ABB RAPID module: SERVER.mod

MODULE SERVER

!////////////////
!GLOBAL VARIABLES
!////////////////

!//Robot configuration
PERS tooldata currentTool := [TRUE,[[0,0,0],[-0.27065,0.65328,-0.2706,0.65328]],[0.001,[0,0,0.001],[1,0,0,0],0,0,0]];
PERS wobjdata currentWobj := [FALSE,TRUE,"",[[0,0,0],[1,0,0,0]],[[0,0,0],[1,0,0,0]]];
PERS speeddata currentSpeed;
PERS zonedata currentZone;

!// Clock Synchronization
PERS bool startLog:=TRUE;
PERS bool startRob:=TRUE;

!// Mutex between logger and changing the tool and work objects
PERS bool frameMutex:=FALSE;

!//PC communication
VAR socketdev clientSocket;
VAR socketdev serverSocket;
VAR num instructionCode;
VAR num params{10};
VAR num nParams;

PERS string ipController:= "20.20.20.21"; !robot default IP
!PERS string ipController:= "127.0.0.1"; !local IP for testing in simulation
PERS num serverPort:= 5000;

!//Motion of the robot
VAR robtarget cartesianTarget;
VAR jointtarget jointsTarget;
VAR bool moveCompleted; !Set to true after finishing a Move instruction.

!//Buffered move variables
CONST num MAX_BUFFER := 128;
PERS bool paused := FALSE;
PERS num BUFFER_POS;
PERS num BUFFER_LEFT;
PERS bool MOVING;
PERS robtarget bufferTargets{MAX_BUFFER};
PERS speeddata bufferSpeeds{MAX_BUFFER};
PERS bool BUFFER_LOCKED;

!//External axis position variables
PERS extjoint externalAxis;

!//Circular move buffer
VAR robtarget circPoint;

!//Correct Instruction Execution and possible return values
VAR num ok;
CONST num SERVER_BAD_MSG :=  0;
CONST num SERVER_OK := 1;




!////////////////
!LOCAL METHODS
!////////////////

!//Method to parse the message received from a PC
!// If correct message, loads values on:
!// - instructionCode.
!// - nParams: Number of received parameters.
!// - params{nParams}: Vector of received params.
PROC ParseMsg(string msg)
    !//Local variables
    VAR bool auxOk;
    VAR num ind:=1;
    VAR num newInd;
    VAR num length;
    VAR num indParam:=1;
    VAR string subString;
    VAR bool end := FALSE;

    !//Find the end character
    length := StrMatch(msg,1,"#");
    IF length > StrLen(msg) THEN
        !//Corrupt message
        nParams := -1;
    ELSE
        !//Read Instruction code
        newInd := StrMatch(msg,ind," ") + 1;
        subString := StrPart(msg,ind,newInd - ind - 1);
        auxOk:= StrToVal(subString, instructionCode);
        IF auxOk = FALSE THEN
            !//Impossible to read instruction code
            nParams := -1;
        ELSE
            ind := newInd;
            !//Read all instruction parameters (maximum of 8)
            WHILE end = FALSE DO
                newInd := StrMatch(msg,ind," ") + 1;
                IF newInd > length THEN
                    end := TRUE;
                ELSE
                    subString := StrPart(msg,ind,newInd - ind - 1);
                    auxOk := StrToVal(subString, params{indParam});
                    indParam := indParam + 1;
                    ind := newInd;
                ENDIF
            ENDWHILE
            nParams:= indParam - 1;
        ENDIF
    ENDIF
ENDPROC


!//Handshake between server and client:
!// - Creates socket.
!// - Waits for incoming TCP connection.
PROC ServerCreateAndConnect(string ip, num port)
    VAR string clientIP;

    SocketCreate serverSocket;
    SocketBind serverSocket, ip, port;
    SocketListen serverSocket;
    TPWrite "SERVER: Server waiting for incoming connections ...";
    WHILE SocketGetStatus(clientSocket) <> SOCKET_CONNECTED DO
        SocketAccept serverSocket,clientSocket \ClientAddress:=clientIP \Time:=WAIT_MAX;
        IF SocketGetStatus(clientSocket) <> SOCKET_CONNECTED THEN
            TPWrite "SERVER: Problem serving an incoming connection.";
            TPWrite "SERVER: Try reconnecting.";
        ENDIF
        !//Wait 0.5 seconds for the next reconnection
        WaitTime 0.5;
    ENDWHILE
    TPWrite "SERVER: Connected to IP " + clientIP;
ENDPROC


!//Parameter initialization
!// Loads default values for
!// - Tool.
!// - WorkObject.
!// - Zone.
!// - Speed.
PROC Initialize()
    currentTool := [TRUE,[[0,0,0],[1,0,0,0]],[0.001,[0,0,0.001],[1,0,0,0],0,0,0]];
    currentWobj := [FALSE,TRUE,"",[[0,0,0],[1,0,0,0]],[[0,0,0],[1,0,0,0]]];
    currentSpeed := [250, 250, 250, 250];
    currentZone := [FALSE, 0.3, 0.3,0.3,0.03,0.3,0.03]; !z0

	!Find the current external axis values so they don't move when we start
	jointsTarget := CJointT();
	externalAxis := jointsTarget.extax;
ENDPROC


!////////////////////////
!//SERVER: Main procedure
!////////////////////////
PROC main()
    !//Local variables
    VAR string receivedString;   !//Received string
    VAR string sendString;       !//Reply string
    VAR string addString;        !//String to add to the reply.
    VAR bool connected;          !//Client connected
    VAR bool reconnected;        !//Drop and reconnection happened during serving a command
    VAR robtarget cartesianPose;
    VAR jointtarget jointsPose;

    VAR robtarget pwobj1;
    VAR robtarget pwobj2;
    VAR robtarget pwobj3;
    VAR wobjdata cwobj;
    VAR num writePos := 1;

    VAR num speed := 250;
    VAR speeddata newSpeed;


    !//Motion configuration
    !ConfL \Off;
    !SingArea \Wrist;
    moveCompleted:= TRUE;

    !//Initialization of WorkObject, Tool, Speed and Zone
    Initialize;

    !//Socket connection
    connected:=FALSE;
    ServerCreateAndConnect ipController,serverPort;
    connected:=TRUE;

    !//Server Loop
    WHILE TRUE DO
        !//Initialization of program flow variables
        ok:=SERVER_OK;              !//Correctness of executed instruction.
        reconnected:=FALSE;         !//Has communication dropped after receiving a command?
        addString := "";

        !//Wait for a command
        SocketReceive clientSocket \Str:=receivedString  \ReadNoOfBytes:=76 \Time:=WAIT_MAX;
        ParseMsg receivedString;

        !//Execution of the command
        TEST instructionCode
            CASE 0: !Ping
                IF nParams = 0 THEN
                    ok := SERVER_OK;
                ELSE
                    ok := SERVER_BAD_MSG;
                ENDIF

!            CASE 1: !Cartesian Move
!                IF nParams = 7 THEN
!                    cartesianTarget :=[[params{1},params{2},params{3}],
!                                       [params{4},params{5},params{6},params{7}],
!                                       [0,0,0,0],
!                                       externalAxis];
!                    ok := SERVER_OK;
!                    moveCompleted := FALSE;
!                    MoveL cartesianTarget, currentSpeed, currentZone, currentTool \WObj:=currentWobj ;
!                    moveCompleted := TRUE;
!                ELSE
!                    ok := SERVER_BAD_MSG;
!                ENDIF

!            CASE 2: !Joint Move
!                IF nParams = 6 THEN
!                    jointsTarget:=[[params{1},params{2},params{3},params{4},params{5},params{6}], externalAxis];
!                    ok := SERVER_OK;
!                    moveCompleted := FALSE;
!                    MoveAbsJ jointsTarget, currentSpeed, currentZone, currentTool \Wobj:=currentWobj;
!                    moveCompleted := TRUE;
!                ELSE
!                    ok :=SERVER_BAD_MSG;
!                ENDIF

            CASE 3: !Get Cartesian Coordinates (with current tool and workobject)
                IF nParams = 0 THEN
                    cartesianPose := CRobT(\Tool:=currentTool \WObj:=currentWObj);
                    addString := NumToStr(cartesianPose.trans.x,2) + " ";
                    addString := addString + NumToStr(cartesianPose.trans.y,2) + " ";
                    addString := addString + NumToStr(cartesianPose.trans.z,2) + " ";
                    addString := addString + NumToStr(cartesianPose.rot.q1,3) + " ";
                    addString := addString + NumToStr(cartesianPose.rot.q2,3) + " ";
                    addString := addString + NumToStr(cartesianPose.rot.q3,3) + " ";
                    addString := addString + NumToStr(cartesianPose.rot.q4,3); !End of string
                    ok := SERVER_OK;
                ELSE
                    ok :=SERVER_BAD_MSG;
                ENDIF

            CASE 4: !Get Joint Coordinates
                IF nParams = 0 THEN
                    jointsPose := CJointT();
                    addString := NumToStr(jointsPose.robax.rax_1,2) + " ";
                    addString := addString + NumToStr(jointsPose.robax.rax_2,2) + " ";
                    addString := addString + NumToStr(jointsPose.robax.rax_3,2) + " ";
                    addString := addString + NumToStr(jointsPose.robax.rax_4,2) + " ";
                    addString := addString + NumToStr(jointsPose.robax.rax_5,2) + " ";
                    addString := addString + NumToStr(jointsPose.robax.rax_6,2); !End of string
                    ok := SERVER_OK;
                ELSE
                    ok:=SERVER_BAD_MSG;
                ENDIF
			CASE 5: !Get external axis positions
                IF nParams = 0 THEN
                    jointsPose := CJointT();
                    addString := StrPart(NumToStr(jointsTarget.extax.eax_a, 2),1,8) + " ";
                    addString := addString + StrPart(NumToStr(jointsTarget.extax.eax_b,2),1,8) + " ";
                    addString := addString + StrPart(NumToStr(jointsTarget.extax.eax_c,2),1,8) + " ";
                    addString := addString + StrPart(NumToStr(jointsTarget.extax.eax_d,2),1,8) + " ";
                    addString := addString + StrPart(NumToStr(jointsTarget.extax.eax_e,2),1,8) + " ";
                    addString := addString + StrPart(NumToStr(jointsTarget.extax.eax_f,2),1,8); !End of string
                    ok := SERVER_OK;
                ELSE
                    ok:=SERVER_BAD_MSG;
                ENDIF

            CASE 6: !Set Tool
                IF nParams = 7 THEN
		   WHILE (frameMutex) DO
		        WaitTime .01; !// If the frame is being used by logger, wait here
		   ENDWHILE
		frameMutex:= TRUE;
                    currentTool.tframe.trans.x:=params{1};
                    currentTool.tframe.trans.y:=params{2};
                    currentTool.tframe.trans.z:=params{3};
                    currentTool.tframe.rot.q1:=params{4};
                    currentTool.tframe.rot.q2:=params{5};
                    currentTool.tframe.rot.q3:=params{6};
                    currentTool.tframe.rot.q4:=params{7};
                    ok := SERVER_OK;
		    frameMutex:= FALSE;
                ELSE
                    ok:=SERVER_BAD_MSG;
                ENDIF

            CASE 7: !Set Work Object
                IF nParams = 7 THEN
                    currentWobj.oframe.trans.x:=params{1};
                    currentWobj.oframe.trans.y:=params{2};
                    currentWobj.oframe.trans.z:=params{3};
                    currentWobj.oframe.rot.q1:=params{4};
                    currentWobj.oframe.rot.q2:=params{5};
                    currentWobj.oframe.rot.q3:=params{6};
                    currentWobj.oframe.rot.q4:=params{7};
                    ok := SERVER_OK;
                ELSE
                    ok:=SERVER_BAD_MSG;
                ENDIF

            CASE 8: !Set Speed of the Robot
                !IF nParams = 4 THEN
                !    currentSpeed.v_tcp:=params{1};
                !    currentSpeed.v_ori:=params{2};
                !    currentSpeed.v_leax:=params{3};
                !    currentSpeed.v_reax:=params{4};
                !    ok := SERVER_OK;
                !ELSEIF nParams = 2 THEN
				!	currentSpeed.v_tcp:=params{1};
				!	currentSpeed.v_ori:=params{2};
				!	ok := SERVER_OK;
				!ELSE
                !    ok:=SERVER_BAD_MSG;
                !ENDIF

            CASE 9: !Set zone data
                IF nParams = 4 THEN
                    IF params{1}=1 THEN
                        currentZone.finep := TRUE;
                        currentZone.pzone_tcp := 0.0;
                        currentZone.pzone_ori := 0.0;
                        currentZone.zone_ori := 0.0;
                    ELSE
                        currentZone.finep := FALSE;
                        currentZone.pzone_tcp := params{2};
                        currentZone.pzone_ori := params{3};
                        currentZone.zone_ori := params{4};
                    ENDIF
                    ok := SERVER_OK;
                ELSE
                    ok:=SERVER_BAD_MSG;
                ENDIF

            CASE 30: !Add Cartesian Coordinates to buffer
                WHILE BUFFER_LOCKED DO
                    !wait
                ENDWHILE
                IF nParams = 8 THEN
                    cartesianTarget :=[[params{1},params{2},params{3}],
                                        [params{4},params{5},params{6},params{7}],
                                        [0,0,0,0],
                                        externalAxis];

                    speed := params{8};
                    if speed < 1 OR speed > 250 THEN
                        newSpeed := [250, 250, 250, 250];
                    ELSE
                        newSpeed := [speed, speed, speed, speed];
                    ENDIF

!                    IF BUFFER_POS < MAX_BUFFER THEN
!                        BUFFER_POS := BUFFER_POS + 1;
!                        bufferTargets{BUFFER_POS} := cartesianTarget;
!                        bufferSpeeds{BUFFER_POS} := newSpeed;
!                    ENDIF
                    IF BUFFER_LEFT > 0 THEN
                        writePos := writePos+1;
                        IF writePos > MAX_BUFFER THEN
                            writePos := writePos - MAX_BUFFER;
                        ENDIF
                        bufferTargets{writePos} := cartesianTarget;
                        bufferSpeeds{writePos} := newSpeed;
                        BUFFER_LEFT := BUFFER_LEFT - 1;
                    ENDIF
                    !addString := NumToStr(MAX_BUFFER - BUFFER_POS,2);
                    addString := NumToStr(BUFFER_LEFT,2);
                    ok := SERVER_OK;
                ELSE
                    ok:=SERVER_BAD_MSG;
                ENDIF

            CASE 31: !Clear Cartesian Buffer
                WHILE BUFFER_LOCKED DO
                    !wait
                ENDWHILE
                IF nParams = 0 THEN
                    writePos := 0;
                    IF MOVING THEN
                        BUFFER_LEFT := MAX_BUFFER - 1;
                        BUFFER_POS := 0;
                    ELSE
                        BUFFER_LEFT := MAX_BUFFER;
                        BUFFER_POS := 1;
                    ENDIF
                    ok := SERVER_OK;
                ELSE
                    ok:=SERVER_BAD_MSG;
                ENDIF

            CASE 32: !Get Buffer Size)
                WHILE BUFFER_LOCKED DO
                    !wait
                ENDWHILE
                IF nParams = 0 THEN
                    addString := NumToStr(MAX_BUFFER-BUFFER_LEFT,2);
                    ok := SERVER_OK;
                ELSE
                    ok:=SERVER_BAD_MSG;
                ENDIF

!            CASE 33: !Execute moves in cartesianBuffer as linear moves
!                IF nParams = 0 THEN
!                    FOR i FROM 1 TO (BUFFER_POS) DO
!                        MoveL bufferTargets{i}, bufferSpeeds{i}, currentZone, currentTool \WObj:=currentWobj ;
!                    ENDFOR
!                    ok := SERVER_OK;
!                ELSE
!                    ok:=SERVER_BAD_MSG;
!                ENDIF

!            CASE 34: !External Axis move
!                IF nParams = 6 THEN
!                    externalAxis :=[params{1},params{2},params{3},params{4},params{5},params{6}];
!                    jointsTarget := CJointT();
!                    jointsTarget.extax := externalAxis;
!                    ok := SERVER_OK;
!                    moveCompleted := FALSE;
!                    MoveAbsJ jointsTarget, currentSpeed, currentZone, currentTool \Wobj:=currentWobj;
!                    moveCompleted := TRUE;
!                ELSE
!                    ok :=SERVER_BAD_MSG;
!                ENDIF

!            CASE 35: !Specify circPoint for circular move, and then wait on toPoint
!                IF nParams = 7 THEN
!                    circPoint :=[[params{1},params{2},params{3}],
!                                [params{4},params{5},params{6},params{7}],
!                                [0,0,0,0],
!                                externalAxis];
!                    ok := SERVER_OK;
!                ELSE
!                    ok:=SERVER_BAD_MSG;
!                ENDIF

!            CASE 36: !specify toPoint, and use circPoint specified previously
!                IF nParams = 7 THEN
!                    cartesianTarget :=[[params{1},params{2},params{3}],
!                                        [params{4},params{5},params{6},params{7}],
!                                        [0,0,0,0],
!                                        externalAxis];
!                    MoveC circPoint, cartesianTarget, currentSpeed, currentZone, currentTool \WObj:=currentWobj ;
!                    ok := SERVER_OK;
!                ELSE
!                    ok:=SERVER_BAD_MSG;
!                ENDIF

            CASE 80:
                !pwobj1 :=[[1400,-655,880],[1,0,0,0],[0,0,0,0],externalAxis];
                !pwobj2 :=[[2180,-655,880],[1,0,0,0],[0,0,0,0],externalAxis];
                !pwobj3 :=[[1400,460,880],[1,0,0,0],[0,0,0,0],externalAxis];
                cwobj := [ FALSE, TRUE, "", [ [0, 0, 0], [1, 0, 0 ,0] ], [ [0, 200, 30], [1, 0, 0 ,0] ] ];
                cwobj.oframe := DefFrame(pwobj1, pwobj2, pwobj3);
                addString := NumToStr(cwobj.oframe.trans.x,2) + " ";
                addString := addString + NumToStr(cwobj.oframe.trans.y,2) + " ";
                addString := addString + NumToStr(cwobj.oframe.trans.z,2) + " ";
                addString := addString + NumToStr(cwobj.oframe.rot.q1,3) + " ";
                addString := addString + NumToStr(cwobj.oframe.rot.q2,3) + " ";
                addString := addString + NumToStr(cwobj.oframe.rot.q3,3) + " ";
                addString := addString + NumToStr(cwobj.oframe.rot.q4,3); !End of string
                TPWrite addString;
                ok := SERVER_OK;

            CASE 81:
                pwobj1 :=[[params{1},params{2},params{3}],[params{4},params{5},params{6},params{7}],[0,0,0,0],externalAxis];
                ok := SERVER_OK;
            CASE 82:
                pwobj2 :=[[params{1},params{2},params{3}],[params{4},params{5},params{6},params{7}],[0,0,0,0],externalAxis];
                ok := SERVER_OK;
            CASE 83:
                pwobj3 :=[[params{1},params{2},params{3}],[params{4},params{5},params{6},params{7}],[0,0,0,0],externalAxis];
                ok := SERVER_OK;


            CASE 90: !pause
                paused := TRUE;
                StopMove;
                ok:=SERVER_OK;

            CASE 91: !resume
                paused := FALSE;
                StartMove;
                ok:=SERVER_OK;

            CASE 98: !returns current robot info: serial number, robotware version, and robot type
                IF nParams = 0 THEN
                    addString := GetSysInfo(\SerialNo) + "*";
                    addString := addString + GetSysInfo(\SWVersion) + "*";
                    addString := addString + GetSysInfo(\RobotType);
                    ok := SERVER_OK;
                ELSE
                    ok :=SERVER_BAD_MSG;
                ENDIF

            CASE 99: !Close Connection
                IF nParams = 0 THEN
                    TPWrite "SERVER: Client has closed connection.";
                    connected := FALSE;
                    !//Closing the server
                    SocketClose clientSocket;
                    SocketClose serverSocket;

                    !Reinitiate the server
                    ServerCreateAndConnect ipController,serverPort;
                    connected := TRUE;
                    reconnected := TRUE;
                    ok := SERVER_OK;
                ELSE
                    ok := SERVER_BAD_MSG;
                ENDIF
            DEFAULT:
                TPWrite "SERVER: Illegal instruction code" + NumToStr(instructionCode,0);
                ok := SERVER_BAD_MSG;
                TPWrite receivedString;
        ENDTEST

        !Compose the acknowledge string to send back to the client
        IF connected = TRUE THEN
            IF reconnected = FALSE THEN
			    IF SocketGetStatus(clientSocket) = SOCKET_CONNECTED THEN
				    sendString := NumToStr(instructionCode,0);
                    sendString := sendString + " " + NumToStr(ok,0);
                    sendString := sendString + " " + addString;
                    !TPWrite sendString;
                    SocketSend clientSocket \Str:=sendString;
			    ENDIF
            ENDIF
        ENDIF
    ENDWHILE

ERROR (LONG_JMP_ALL_ERR)
    TPWrite "SERVER: ------";
    TPWrite "SERVER: Error Handler:" + NumtoStr(ERRNO,0);
    TEST ERRNO
        CASE ERR_SOCK_CLOSED:
            TPWrite "SERVER: Lost connection to the client.";
            TPWrite "SERVER: Closing socket and restarting.";
            TPWrite "SERVER: ------";
            connected:=FALSE;
            !//Closing the server
            SocketClose clientSocket;
            SocketClose serverSocket;
            !//Reinitiate the server
            ServerCreateAndConnect ipController,serverPort;
            reconnected:= FALSE;
            connected:= TRUE;
            RETRY;
        DEFAULT:
            TPWrite "SERVER: Unknown error.";
            TPWrite "SERVER: Closing socket and restarting.";
            TPWrite "SERVER: ------";
            connected:=FALSE;
            !//Closing the server
            SocketClose clientSocket;
            SocketClose serverSocket;
            !//Reinitiate the server
            ServerCreateAndConnect ipController,serverPort;
            reconnected:= FALSE;
            connected:= TRUE;
            RETRY;
    ENDTEST
ENDPROC

ENDMODULE
